VAR_GLOBAL
////////////////////////////////////////:	///////////////////////////////////////////////////
/////////////////////////////////////////////////////////////////////////////////////GENERIC/////////////////////////////////////////////////////////////////////////////////////

	bQuitHMI							: BOOL;
	bShutDown							: BOOL;
	stStatusBanner						: ST_StatusBanner;
	nPopUp								: DINT;
	
	bPartPresent						: ARRAY [0..1] OF BOOL;
	
	bRejectPartDialog					: ARRAY [0..2] OF BOOL;
	bOpenRejectDialog					: BOOL;
	anCameraScore						: ARRAY [1..2] OF STRING;
	bLightsOnOff						: BOOL;
	
	bHMIAlive							: BOOL;
	tonHMIAliveOn						: TON;
	tonHMIAliveOff						: TON;
	bOutHMI								: BOOL;
	bEmptyRejectChuteAcknowledge  		: BOOL;
	bEmptyRejectChute					: BOOL;
	bSavePersistentData					: BOOL;
	
/////////////////////////////////////////////////////////////////////////////////////SYSTEM INFO/////////////////////////////////////////////////////////////////////////////////////

	sSoftwareVersion					: STRING := ' v1.0.0-rc.2';
	sSoftwareDate						: STRING := '03/08/2026';
	sTC3Version							: STRING := ' v3.1.4026.22, Runtime v3.1.4026.22 ';
	sHMIVersion							: STRING := ' 14.13';
	sSystemName							: STRING := 'LT-WH-VC Serter';
	sProjectID							: STRING := ' TE 11108' ;
	sAplication                     	: STRING ;
	sHMIServer                			: STRING := ' 14.13 ';
	
/////////////////////////////////////////////////////////////////////////////////////MANUAL/////////////////////////////////////////////////////////////////////////////////////

	bEnableManual						: BOOL;
	nMainRegion							: DINT;
	bManualModeOffFlag					: BOOL;
	bManualScreen						: BOOL;
	tonManualMode						: TON;
	bEnableSettings						: BOOL;
			
	bProcessDoor_Up						: BOOL;
	bProcessDoor_Down					: BOOL;

	bLeaktester1_Start					: BOOL;
	bLeaktester2_Start					: BOOL;
	bLeaktester1_Stop					: BOOL;
	bLeaktester2_Stop					: BOOL;
	bLeaktester1_Reset					: BOOL;
	bLeaktester2_Reset					: BOOL;
	
	bCameraResetStatistics				: ARRAY[1..2] OF BOOL;
	bCameraSettingNo					: ARRAY[1..2] OF UINT;
	bCameraSettingVal					: ARRAY[1..2] OF UDINT;
	bCameraSetTreshold					: ARRAY[1..2] OF BOOL;
	bCameraTrigger						: ARRAY[1..2] OF BOOL;
	
	bProcessCtlinderExtend1				: BOOL;
	bProcessCtlinderRetract1			: BOOL;
	bProcessCtlinderExtend2				: BOOL;
	bProcessCtlinderRetract2			: BOOL;
	
	bHoldPart1							: BOOL;
	bHoldPart2							: BOOL;
	
	bVacuumCylinderExtend1				: BOOL;
	bVacuumCylinderRetract1				: BOOL;
	bVacuumCylinderExtend2				: BOOL;
	bVacuumCylinderRetract2				: BOOL;
	
	bPartHeld							: ARRAY[1..2] OF BOOL;
	
	bEnable_ProcessCylinder				: ARRAY[1..2] OF BOOL;
	bEnable_VacuumCylinder				: ARRAY[1..2] OF BOOL;
	bEnable_Holder						: ARRAY[1..2] OF BOOL;
	
	bSetCalibrationHeight1				: BOOL;
	bSetCalibrationHeight2				: BOOL;
	
	bTriggerLSS							: BOOL;
	
	(*Renan Added - 06Jul26 - Getting offset from HMI*)
	//Puck Locker
	stPuckLocker 						: ST_PuckLockerHMI;
	(*\Renan Added - 06Jul26 - Getting offset from HMI*)
	
	
	
	
END_VAR

VAR_GLOBAL PERSISTENT
	
	stTimers							: ST_Timers;
	stStatisticsHMI						: ARRAY [0..7] OF ST_StatisticsHMI;	//0: Nest1
																	//1: Nest2
																	//2: Leak Tester 1
																	//3: Leak Tester 2
																	//4: Height Check 1
																	//5: Height Check 2
																	//6: Vision Check 1
																	//7: Vision Check 2
																	
																	
														
	/////////////////////////////////////////////////////////////////////////////////////SETTINGS/////////////////////////////////////////////////////////////////////////////////////	


	(*Renan Added - 06Jul26 - Getting offset from HMI*)
	ePuckLockerMode : E_PuckLockerMode := E_PuckLockerMode.Disabled; //Puck locker state
	bPuckLockerGateEnable 				: BOOL := TRUE;
	bPuckLockerSkipEnable 				: BOOL := FALSE;
	(*\Renan Added - 06Jul26 - Getting offset from HMI*)
	
	
	//TwinSAFE
	
	nAirPressureMaxValue				: UINT;	
	nAirPressureMinValue				: UINT;	
	
	bNest1Flag							: BOOL;
	bNest2Flag							: BOOL;
	
	nHeightSetByCalibration				: REAL;
	nHeightTolerance					: REAL;
	nHeightSetPoint						: REAL;


	
END_VAR

(* stored: Version 1.1.0.1, ProductVersion 3.1.4026.18
   GVL GVL_HMI: Id {7d424ba3-5d42-48e0-870b-7d749b127bab} *)
